# EPICS autosave request: iocBoot/iocTomoScan_19BM/auto_settings.req
file "tomoScan_settings.req", P=$(P), R=$(R)
file "tomoScan_PSO_settings.req", P=$(P), R=$(R)
file "tomoScan_19BM_settings.req", P=$(P), R=$(R)
